FUNCTION_BLOCK FB_ModbusMaster //IMPLEMENTS I_UniversalUnit
VAR
	sName			:		STRING;
	bInitialized	:		BOOL;
	iScantime		:		UINT;
	iTimeout		:		UINT := 1000;//1000ms
	iErrorID		:		MODBUS_ERRORS;
	bBusy			: 		BOOL;
	bError			:		BOOL;
	iStepGeneral	: 		E_ModBusMasterState;
	iStepRunning	:		E_ModbusMasterStateRun;
	bFirstCycle		:		BOOL;
	bRun			:		BOOL;
	bStop			: 		BOOL;

	fbModbusMaster	: 		ModbusRtuMaster_PcCOM;
	//fbModbusMaster : 		ModbusRtuMasterV2_KL6x22B;
	ipModbusSlave	:		ARRAY [1..247] OF I_ModbusSlave;
	iAmountSlave	: 		UINT;
	
	iLoopSlave		:		UINT	:= 1;
	iLoopAdr		:		UINT;
	iQuantity 		: 		POINTER TO WORD;
	iMBAddr 		: 		POINTER TO WORD;
    arrData			: 		ARRAY [0..255] OF WORD;
	
	UnitId	: BYTE;
	Quantity	: WORD;
	MBAddr	: WORD;
	cbLength : UINT;
	pMemoryAddr	: POINTER TO BYTE;
	pDataWrite	: POINTER TO WORD;

	bexecute	: BOOL;
	
	tCalculateTimeRW	: TON;
	nNumberFaultRW	: UINT;
	eModbusFunction: E_ModbusFunction;
	peModbusFunction : POINTER TO WORD;
END_VAR

StateMachine();
bRun :=  iStepGeneral = E_ModBusMasterState.Running ;
bStop := iStepGeneral = E_ModBusMasterState.stop_done;
bInitialized := iStepGeneral >= E_ModBusMasterState.Ready;
iErrorID := fbModbusMaster.ErrorId;
tCalculateTimeRW(PT	:= T#10S); // for test how much time read write total

METHOD Abort : BOOL
bError := FALSE;
iErrorID := 0;
bError := FALSE;
iStepGeneral	:= E_ModBusMasterState.Uninitialized;
iStepRunning	:= E_ModbusMasterStateRun.CheckNumberSlaveRegistered;

iLoopSlave		:= 1;
iLoopAdr		:= 0;

fbModbusMaster(Execute := FALSE);

Abort := TRUE;
END_METHOD

PROPERTY AnyError : BOOL
GET
AnyError 	:= bError;
END_GET
END_PROPERTY

PROPERTY Busy : BOOL
GET
Busy := bBusy;
END_GET
END_PROPERTY

PROPERTY ErrorID : MODBUS_ERRORS
GET
ErrorID := iErrorID;
END_GET
END_PROPERTY

METHOD Init : BOOL
IF iStepGeneral = E_ModBusMasterState.Uninitialized THEN
	iStepGeneral := E_ModBusMasterState.Initializing;
END_IF

//Method output
	Init := (iStepGeneral >= E_ModBusMasterState.Ready);
END_METHOD

PROPERTY Initialized : BOOL
GET
Initialized := bInitialized;
END_GET
END_PROPERTY

PROPERTY Name : STRING
GET
Name := sName;
END_GET
SET
sName := Name;
END_SET
END_PROPERTY

PROPERTY ReadData : ARRAY [0..255] OF Word
GET
ReadData := arrData;
END_GET
END_PROPERTY

PROPERTY ReadDataSize : uint
GET
ReadDataSize := INT_TO_UINT(SIZEOF(arrData));
END_GET
END_PROPERTY

METHOD RegisterSlave : BOOL
VAR_INPUT
	ModbusSlave		:		I_ModbusSlave;
END_VAR
VAR
	iLoop	:	UINT;
	bExists	:	BOOL;
END_VAR
FOR iLoop := 1 TO iAmountSlave DO
	IF ipModbusSlave[iLoop] = ModbusSlave THEN
		bExists := TRUE;
		iLoop := iAmountSlave;// end loop for command
	END_IF
END_FOR 
IF NOT bExists THEN
	iAmountSlave := iAmountSlave + 1;
	ipModbusSlave[iAmountSlave] := ModbusSlave;
END_IF
END_METHOD

METHOD Reset : BOOL
bError := FALSE;
iErrorID := 0;
bError := FALSE;
iStepGeneral	:= E_ModBusMasterState.Uninitialized;
iStepRunning	:= E_ModbusMasterStateRun.CheckNumberSlaveRegistered;

iLoopSlave		:= 1;
iLoopAdr		:= 0;

fbModbusMaster.Execute := FALSE;

Reset := TRUE;
END_METHOD

METHOD Run : BOOL /// call from FB_modbus
IF (iStepGeneral = E_ModBusMasterState.Ready) THEN
	iStepGeneral := E_ModBusMasterState.Running;
END_IF

bRun := TRUE;
Run := (iStepGeneral >= E_ModBusMasterState.Running) AND (iStepGeneral < E_ModBusMasterState.stop);
END_METHOD

PROPERTY ScanTime : UINT
GET
ScanTime := iScantime;
END_GET
SET
iScantime := ScanTime;
END_SET
END_PROPERTY

METHOD protected StateInit : BOOL (*Unit is performing initialization*)
IF NOT bError THEN
	iStepGeneral := E_ModBusMasterState.Ready;
END_IF
END_METHOD

METHOD protected StateMachine : BOOL (*State machine of unit*)
CASE iStepGeneral OF
		E_ModBusMasterState.Uninitialized:  
			StateUninitialized();
	
		E_ModBusMasterState.Initializing: 
			StateInit();
	
		E_ModBusMasterState.Ready: 
			StateReady();
		
		E_ModBusMasterState.Running: 
			StateRunning();
						
		E_ModBusMasterState.stop:
			StateStopping();
			
		E_ModBusMasterState.stop_done:
			StateStoppingDone();
END_CASE
END_METHOD

METHOD protected StateReady : BOOL (* Unit is initialized*)
END_METHOD

METHOD PROTECTED StateRunning : BOOL (* Unit is uninitialized*)
VAR 
	

	
END_VAR
CASE iStepRunning OF
	E_ModbusMasterStateRun.CheckNumberSlaveRegistered: // Trigger
		IF iAmountSlave > 0 THEN
			iStepRunning := E_ModbusMasterStateRun.SetParametersRead;
		END_IF
					
	E_ModbusMasterStateRun.SetParametersRead: // Set parameters
		IF ipModbusSlave[iLoopSlave].NumAddRegionRead <> 0 
		AND iLoopAdr <= (ipModbusSlave[iLoopSlave].NumAddRegionRead - 1) 
		THEN
			iQuantity := ipModbusSlave[iLoopSlave].AddressRead + ((iLoopAdr * 3 + 1) * SIZEOF(WORD));// arrAddressRead[iloopAdr][1] in Slave
			iMBAddr := ipModbusSlave[iLoopSlave].AddressRead + ((iLoopAdr * 3) * SIZEOF(WORD));// arrAddressRead[iloopAdr][0] in Slave
			UnitID := ipModbusSlave[iLoopSlave].UnitID;
			Quantity :=	iQuantity^;
			MBAddr := iMBAddr^;
			cbLength := SIZEOF(arrData);
			pMemoryAddr	:= ADR(arrData);
			peModbusFunction := ipModbusSlave[iLoopSlave].AddressRead + ((iLoopAdr * 3 + 2) * SIZEOF(WORD)); // arrAddressRead[iloopAdr][2] in Slave
			eModbusFunction := peModbusFunction^;
			iStepRunning := E_ModbusMasterStateRun.SendRequestRead;
		ELSE 
			iLoopAdr := 0;
			iStepRunning := E_ModbusMasterStateRun.ReturnReadDone;
		END_IF

			
	E_ModbusMasterStateRun.SendRequestRead: // Send request
		CASE eModbusFunction OF
			E_ModbusFunction.ReadHoldingRegisters:
				fbModbusMaster.ReadRegs(
					UnitID:= UnitID, 
					Quantity:= Quantity, 
					MBAddr:= MBAddr, 
					cbLength:= cbLength, 
					pMemoryAddr:= pMemoryAddr, 
					Execute:= TRUE,
					Timeout:= UINT_TO_TIME(iTimeout),
					BUSY=> bBusy, 
					Error=> bError , 
					ErrorId=>iErrorId 
				);
			
			E_ModbusFunction.ReadInputRegisters:
				fbModbusMaster.ReadInputRegs(
					UnitID:= UnitID, 
					Quantity:= Quantity, 
					MBAddr:= MBAddr, 
					cbLength:= cbLength, 
					pMemoryAddr:= pMemoryAddr, 
					Execute:= TRUE,
					Timeout:= UINT_TO_TIME(iTimeout),
					BUSY=> bBusy, 
					Error=> bError , 
					ErrorId=>iErrorId 
				);
			
		END_CASE
		iStepRunning := E_ModbusMasterStateRun.WaitReadRespond;
						
	E_ModbusMasterStateRun.WaitReadRespond:
		fbModbusMaster.ReadRegs(Execute := FALSE);
		fbModbusMaster.ReadInputRegs(Execute := FALSE);
		ipModbusSlave[iLoopSlave].ModbusErrorID := iErrorID;
		IF NOT fbModbusMaster.BUSY AND NOT fbModbusMaster.Error THEN
			iStepRunning := E_ModbusMasterStateRun.ConvertRawData;
			nNumberFaultRW := 0;
		END_IF
		
		IF fbModbusMaster.Error AND NOT fbModbusMaster.BUSY THEN
			iStepRunning := E_ModbusMasterStateRun.ReturnReadDone;
		END_IF
	
	E_ModbusMasterStateRun.ConvertRawData: 
		ipModbusSlave[iLoopSlave].Convert(
			iRegionNo := iLoopAdr,
		 	pReadData := ADR(arrData)
		);
		iLoopAdr := iLoopAdr + 1;
		iStepRunning := E_ModbusMasterStateRun.CheckNumberSlaveRegistered;

	E_ModbusMasterStateRun.ReturnReadDone: // Return, done
		iStepRunning := E_ModbusMasterStateRun.SetParametersWrite;
		iLoopAdr := 0;

	E_ModbusMasterStateRun.SetParametersWrite :
		IF  ipModbusSlave[iLoopSlave].NumAddRegionWrite <> 0
		AND iLoopAdr <= ipModbusSlave[iLoopSlave].NumAddRegionWrite - 1 
		THEN // iLoopAdr start from 1
			iMBAddr := ipModbusSlave[iLoopSlave].AddressWrite + (iLoopAdr * 11 * SIZEOF(WORD));// return address word contain value address( modbus) 
			pDataWrite := ipModbusSlave[iLoopSlave].AddressWrite + ((iLoopAdr * 11 + 2) * SIZEOF(WORD));
			iQuantity := ipModbusSlave[iLoopSlave].AddressWrite + ((iLoopAdr * 11 + 1) * SIZEOF(WORD));
			peModbusFunction := ipModbusSlave[iLoopSlave].AddressWrite + ((iLoopAdr * 11 + 10) * SIZEOF(WORD));
			eModbusFunction := peModbusFunction^;
			UnitID 	:=		ipModbusSlave[iLoopSlave].UnitID;
			Quantity	:=	iQuantity^;
			MBAddr	:=		iMBAddr^;
			cbLength	:= 	Quantity * 2;
			pMemoryAddr	:= 	pDataWrite;
			iStepRunning := E_ModbusMasterStateRun.SendRequestWrite;
		ELSE 
			iStepRunning := E_ModbusMasterStateRun.ReturnWriteDone;
		END_IF

	E_ModbusMasterStateRun.SendRequestWrite :
		CASE eModbusFunction OF
			E_ModbusFunction.WriteMultipleCoils:
				fbModbusMaster.WriteMultipleCoils(
					UnitID:= UnitID, 
					Quantity:= Quantity, 
					MBAddr:= MBAddr, 
					cbLength:= cbLength, 
					pMemoryAddr:= pMemoryAddr, 
					Execute:=  true,
					Timeout:= 	UINT_TO_TIME(iTimeout),	
					BUSY=> bBusy, 
					Error=> bError , 
					ErrorId=>iErrorId 
				);
													
			E_ModbusFunction.WriteMultipleRegisters:
				fbModbusMaster.WriteRegs(
					UnitID:= UnitID, 
					Quantity:= Quantity, 
					MBAddr:= MBAddr, 
					cbLength:= cbLength, 
					pMemoryAddr:= pMemoryAddr, 
					Execute:= TRUE,
					Timeout:= UINT_TO_TIME(iTimeout),	
					BUSY=> bBusy, 
					Error=> bError , 
					ErrorId=>iErrorId 
				);
											
			E_ModbusFunction.WriteSingleCoil:
				fbModbusMaster.WriteSingleCoil(
					UnitID:= UnitID, 
					Quantity:= Quantity, 
					MBAddr:= MBAddr, 
					cbLength:= cbLength, 
					pMemoryAddr:= pMemoryAddr, 
					Execute:=  true,
					Timeout:= UINT_TO_TIME(iTimeout),	
					BUSY=> bBusy, 
					Error=> bError , 
					ErrorId=>iErrorId 
				);
			E_ModbusFunction.WriteSingleRegister:
				fbModbusMaster.WriteSingleRegister(
					UnitID:= UnitID, 
					Quantity:= Quantity, 
					MBAddr:= MBAddr, 
					cbLength:= cbLength, 
					pMemoryAddr:= pMemoryAddr, 
					Execute:=  true,
					Timeout:= 	UINT_TO_TIME(iTimeout),	
					BUSY=> bBusy, 
					Error=> bError , 
					ErrorId=>iErrorId 
				);
		END_CASE
		
		iStepRunning := E_ModbusMasterStateRun.WaitWriteRespond;
	
	E_ModbusMasterStateRun.WaitWriteRespond :
		fbModbusMaster.WriteMultipleCoils( Execute := FALSE);
		fbModbusMaster.WriteRegs( Execute := FALSE);
		fbModbusMaster.WriteSingleCoil( Execute := FALSE);	
		fbModbusMaster.WriteSingleRegister( Execute := FALSE);
		ipModbusSlave[iLoopSlave].ModbusErrorID := iErrorID;
		IF NOT fbModbusMaster.BUSY AND NOT fbModbusMaster.Error THEN
			iStepRunning := E_ModbusMasterStateRun.SetParametersWrite;
			nNumberFaultRW := 0;
			iLoopAdr := iLoopAdr + 1;
		END_IF
		IF fbModbusMaster.Error AND NOT fbModbusMaster.BUSY THEN
			iStepRunning := E_ModbusMasterStateRun.ReturnWriteDone ;
		END_IF
	
	 E_ModbusMasterStateRun.ReturnWriteDone :
		iLoopAdr := 0;
		iLoopSlave := iLoopSlave + 1;// next slave
		IF iLoopSlave > iAmountSlave THEN
			iLoopSlave := 1;
		END_IF
		THIS^.tCalculateTimeRW(in := FALSE);
		tCalculateTimeRW(in := TRUE);
		iStepRunning := E_ModbusMasterStateRun.CheckNumberSlaveRegistered;
		
END_CASE
END_METHOD

METHOD protected StateStopping : BOOL (* Unit is uninitialized*)
iStepGeneral	:= E_ModBusMasterState.Uninitialized;
iStepRunning	:= E_ModbusMasterStateRun.notKnow;

iLoopSlave		:= 1;
iLoopAdr		:= 0;

fbModbusMaster(Execute := FALSE);
END_METHOD

METHOD protected StateStoppingDone : BOOL (* Unit is uninitialized*)
IF NOT bStop THEN
	iStepGeneral := E_ModBusMasterState.Ready;
END_IF
END_METHOD

METHOD protected StateUninitialized : BOOL (* Unit is uninitialized*)
END_METHOD

METHOD protected Stop : BOOL
IF iStepGeneral >= E_ModBusMasterState.Running AND iStepGeneral < E_ModBusMasterState.stop THEN
	iStepGeneral := E_ModBusMasterState.stop;
END_IF
bStop := TRUE;

Stop := (iStepGeneral = E_ModBusMasterState.stop_done);
END_METHOD

PROPERTY Timeout : UINT // in milisecond, if not respond in this time , error will raise
GET
Timeout := iTimeout;
END_GET
SET
iTimeout := Timeout;
END_SET
END_PROPERTY

END_FUNCTION_BLOCK

(* stored: Version 1.1.0.1, ProductVersion 3.1.4024.12
   POU FB_ModbusMaster: Id {e19cf191-99a0-453d-bfd1-d606b54fb348}, SpecialFunc None
   Folder Methods: Id {322c9666-4625-4231-8f2e-1068372fd37f}
   Folder Property: Id {ba48ab76-59bc-4f33-be02-656bf548ecf8}
   Folder StateMachine: Id {a10f3ecc-db54-4beb-bea9-9e971db1fa22}
   Method Abort: Id {ba4a13e4-31e9-4bb4-bf74-047a8fa89943}
   Property AnyError: Id {f43542ad-5bad-47cb-836f-2409d3407f45}
   Get Get: Id {99e8c5a8-0bce-4e5d-ab0e-0c78eeaaa8db}
   Property Busy: Id {ce498d81-0e66-4915-92c6-32714057e5f8}
   Get Get: Id {fecc03b6-907d-48ef-a4e8-13a5dbedc2e5}
   Property ErrorID: Id {97866986-8d19-4e08-af50-bf6b3ef0a379}
   Get Get: Id {e9f1ee3b-39bf-41e6-9da3-2aecb7d7081f}
   Method Init: Id {306fce68-aa0d-4371-8644-707720662860}
   Property Initialized: Id {bc713903-57dc-4cc6-8f2f-1f1f694f04fb}
   Get Get: Id {5f5f1c81-14c6-419e-8fac-ab921e7efe26}
   Property Name: Id {f7064ea3-a8ae-4c71-9574-c68eee4e83c6}
   Get Get: Id {7f51094e-d0f4-4392-b366-9a5b65b15eec}
   Set Set: Id {4ff50fb1-3d5e-4599-96f4-4237188cd78a}
   Property ReadData: Id {08142e40-5bae-4e54-8781-b37ab4723df3}
   Get Get: Id {1fd5bc5b-9f87-4c50-b2c0-4b04b10d2036}
   Property ReadDataSize: Id {97b1e91b-d519-408b-84bd-bf8d8c70f720}
   Get Get: Id {fa986ddc-918b-40ad-81c5-b83651fe1156}
   Method RegisterSlave: Id {8edb6911-17a5-408b-be71-e6bcb316e950}
   Method Reset: Id {821f3fd7-5ce8-4598-9e42-040f8dab54ce}
   Method Run: Id {216a50ed-05a5-48ba-ace0-07f3271f4b43}
   Property ScanTime: Id {5fc9ff6b-6ff6-4b9f-a579-fafa4fd28c5a}
   Get Get: Id {1d371870-7936-48fa-9375-b3b8dd47659a}
   Set Set: Id {c62ae84c-c593-4921-bc7e-f6479a6e96d6}
   Method StateInit: Id {1349f19a-ff00-4941-afc6-2596d8f2b743}
   Method StateMachine: Id {15a81b95-fbb0-4c76-b869-67165c4df2da}
   Method StateReady: Id {8e715230-e076-4d5e-bf00-f264282f1fe6}
   Method StateRunning: Id {ee25dbd7-315c-4711-865e-cd380d8cdb02}
   Method StateStopping: Id {77b4ba61-0308-4e5b-9ee4-459729c49459}
   Method StateStoppingDone: Id {8e452b4c-ee5a-4ddf-b191-bb7f945b756b}
   Method StateUninitialized: Id {df7bc221-1984-4d12-884a-22de370d4a2b}
   Method Stop: Id {fcc12cb8-f158-41a0-bbc1-7779722b4738}
   Property Timeout: Id {c11aa6a0-86ed-430a-a5cd-d0bbcf967bf2}
   Get Get: Id {0d7eb0fb-ff1a-4356-80f7-df8c23ae0301}
   Set Set: Id {8ad971c0-bc7e-48cb-84b6-163cdabaa78f} *)
